FUNCTION_BLOCK FlushCdt_HMI (* Service Interface Function Block Type *)
  (* Standard: 61499-2 *)
  (* Version 0.0, 6/7/2026, Schneider Electric, template *)
  PACKAGE SE.Nereda;
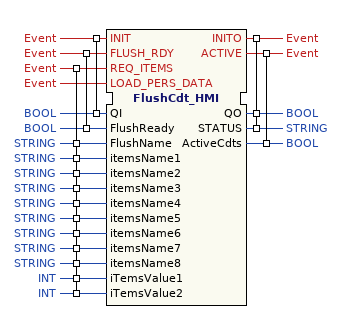
  EVENT_INPUT
    INIT WITH QI;
    FLUSH_RDY WITH FlushReady;
    REQ_ITEMS WITH itemsName1, itemsName2, itemsName3, itemsName4, itemsName5, itemsName6, itemsName7, itemsName8, iTemsValue1, iTemsValue2, FlushName;
    LOAD_PERS_DATA;
  END_EVENT
  EVENT_OUTPUT
    INITO WITH QO, STATUS;
    ACTIVE WITH ActiveCdts;
  END_EVENT
  VAR_INPUT
    QI : BOOL;
    FlushReady : BOOL;
    FlushName : STRING;
    itemsName1 : STRING;
    itemsName2 : STRING;
    itemsName3 : STRING;
    itemsName4 : STRING;
    itemsName5 : STRING;
    itemsName6 : STRING;
    itemsName7 : STRING;
    itemsName8 : STRING;
    iTemsValue1 : INT;
    iTemsValue2 : INT;
  END_VAR
  VAR_OUTPUT
    QO : BOOL; (* Event Output Qualifier *)
    STATUS : STRING; (* Service Status *)
    ActiveCdts : BOOL;
  END_VAR
  SERVICE /
    SEQUENCE 
    END_SEQUENCE
  END_SERVICE
END_FUNCTION_BLOCK
